INTERFACE ITF_TopElement2_HMI_Init EXTENDS ITF_BaseTopElement, ITF_TopElement2_HMI_Connector

END_INTERFACE

(* stored: Version 1.1.0.1, ProductVersion 3.1.4024.15
   Itf ITF_TopElement2_HMI_Init: Id {98df8073-a59f-4119-879d-a2cbc8a8cf16} *)
